PROGRAM P3_08_OpenReport
VAR
	sDateTime			:STRING;
	sYear				:STRING;
	sMonth				:STRING;
	sDay				:STRING;
	sHour				:STRING;
	sMinute				:STRING;
	sReportSuffix		:STRING;
END_VAR

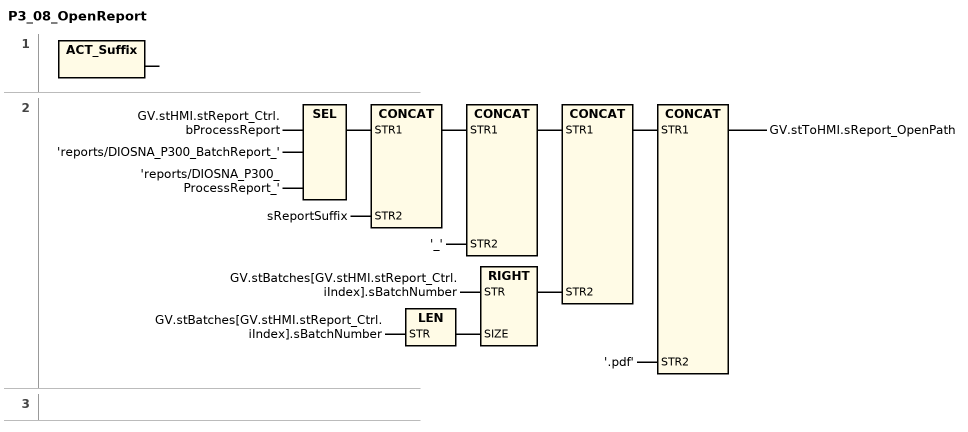
// NETWORK 1
ACT_Suffix();

// NETWORK 2
GV.stToHMI.sReport_OpenPath := CONCAT(STR1 := CONCAT(STR1 := CONCAT(STR1 := CONCAT(STR1 := SEL(GV.stHMI.stReport_Ctrl.bProcessReport, 'reports/DIOSNA_P300_BatchReport_', 'reports/DIOSNA_P300_ProcessReport_'), STR2 := sReportSuffix), STR2 := '_'), STR2 := RIGHT(STR := GV.stBatches[GV.stHMI.stReport_Ctrl.iIndex].sBatchNumber, SIZE := LEN(STR := GV.stBatches[GV.stHMI.stReport_Ctrl.iIndex].sBatchNumber))), STR2 := '.pdf');

// NETWORK 3

ACTION ACT_Suffix:
sDateTime:=GV.stBatches[GV.stHMI.stReport_Ctrl.iIndex].sFinished;
sYear:=RIGHT(LEFT(sDateTime,10),2);
sMonth:=RIGHT(LEFT(sDateTime,5),2);
sDay:=LEFT(sDateTime,2);

sHour:=LEFT(RIGHT(sDateTime,8),2);
sMinute:=LEFT(RIGHT(sDateTime,5),2);

sReportSuffix:=CONCAT(sYear,sMonth);
sReportSuffix:=CONCAT(sReportSuffix,sDay);
sReportSuffix:=CONCAT(sReportSuffix,sHour);
sReportSuffix:=CONCAT(sReportSuffix,sMinute);
END_ACTION

END_PROGRAM

(* stored: Version 1.1.0.1, ProductVersion 3.1.4026.13
   POU P3_08_OpenReport: Id {1b0a9289-824a-4b2f-ad25-6e3ab1574d08}, SpecialFunc None
   Action ACT_Suffix: Id {26e3582a-e3bc-4dbc-83d9-44855f6c4193} *)
